FUNCTION_BLOCK AND_550FE6D62F509EB3 (* Logical AND *)
  (* Standard: 61499-2 *)
  (* Version 1.0, 24.09.2008, marumil, nxtControl GmbH, Initial Version *)
  PACKAGE Main;
  (* Compiler Cpp *)
  {SET_ATTRIBUTE(Runtime.FBType.ImplementingType, Runtime.Standard#DYNGEN_AND)}
  {SET_ATTRIBUTE(Configuration.GenericFBType.InterfaceParams, Runtime.Standard#CNT:=3;OUT:BOOL)}
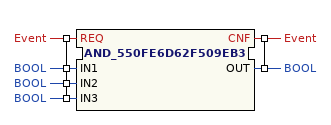
  EVENT_INPUT
    REQ WITH IN1, IN2, IN3; (* Normal Execution Request *)
  END_EVENT
  EVENT_OUTPUT
    CNF WITH OUT; (* Execution Confirmation *)
  END_EVENT
  VAR_INPUT
    IN1 : BOOL; (* Argument *)
    IN2 : BOOL; (* Argument *)
    IN3 : BOOL; (* Argument *)
  END_VAR
  VAR_OUTPUT
    OUT : BOOL; (* Result: IN1 AND IN2 AND ... *)
  END_VAR
  EC_STATES
    START;
  END_STATES
END_FUNCTION_BLOCK
